(* Logix 5000 project; controller PRU vendor 1 type 14 code 107 rev 20.13; software revision 20.01; part 14 of 17 *)
(* tags used below, declared in another part *)
   AlarmMaster : DINT;
   CHANGING_TOTE_1 : BOOL;
   CSS_Status_Data : PLCStatusData;
   DailyTotalResetPB : BOOL;
   GTL1_PRESSURE_Real : REAL;
   GTL1_TEMPERATURE : DINT;
   GTL2_PRESSURE_Real : REAL;
   GTL2_TEMPERATURE : DINT;
   GTL3_PRESSURE_Real : REAL;
   GTL3_TEMPERATURE : DINT;
   IFS_CommsLoss_TMR : TIMER;   // Comms to IFS Has been Lost Alarm Timer
   IFS_CommsLossAlm : BOOL;   // Comms to IFS Has been Lost Alarm
   IFS_CommsWarning_TMR : TIMER;   // Comms to IFS Has been Lost Warning Timer
   IFS_CommsWarningAlm : BOOL;   // Comms to IFS Has been Lost Warning Alarm
   IFS_PLC_Seconds_Temp : DINT;
   IFS_Status_Data : PLCStatusData;
   IND560_Data_to_Set : SINT;
   IND560_Get_Shared_Data_Message : MESSAGE;
   IND560_Read_Data : REAL;
   IND560_Set_Shared_Data_Message : MESSAGE;
   IND560_Test_Msg : MESSAGE;
   KPI_WeightResetPB : BOOL;
   KPI_WeightResetTmr : TIMER;
   LOCAL_DATE_TIME : DateTime;
   MIDNIGHT : BOOL;
   MIDNIGHT_ONS : DINT;
   myweight_2 : DINT;
   myweight_3 : DINT;
   myweight_4 : DINT;
   OutFeedScale : SystemAlarmMonitor;
   PLC_Time : DINT[8];
   PROCESSOR_FAULT : BOOL;
   PRU_Status_Data : PLCStatusData;
   UTL_CommsLoss_TMR : TIMER;   // Comms to UTL Has been Lost Alarm Timer
   UTL_CommsLossAlm : BOOL;   // Comms to UTL Has been Lost Alarm
   UTL_CommsWarning_TMR : TIMER;   // Comms to UTL Has been Lost Warning Timer
   UTL_CommsWarningAlm : BOOL;   // Comms to UTL Has been Lost Warning Alarm
   UTL_PLC_Seconds_Temp : DINT;
   UTL_Status_Data : PLCStatusData;
   WC025_DailyTotal : REAL;
   WC025_DailyTotalLast : REAL;
   WC025_DailyTotalResetPB_ONS : BOOL;
   WC025_TareALM : BOOL;
   WEIGHT : REAL;
(* MSG, continued *)

ROUTINE IFS_MSG   (* ladder *)
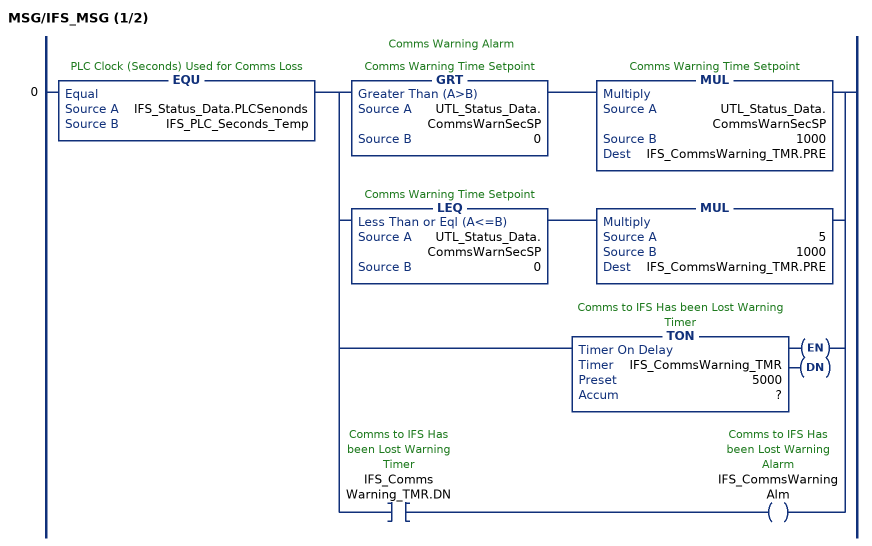
   // Comms Warning Alarm
   0: EQU(IFS_Status_Data.PLCSenonds,IFS_PLC_Seconds_Temp)[GRT(UTL_Status_Data.CommsWarnSecSP,0) MUL(UTL_Status_Data.CommsWarnSecSP,1000,IFS_CommsWarning_TMR.PRE) ,LEQ(UTL_Status_Data.CommsWarnSecSP,0) MUL(5,1000,IFS_CommsWarning_TMR.PRE) ,TON(IFS_CommsWarning_TMR,?,?) ,XIC(IFS_CommsWarning_TMR.DN) OTE(IFS_CommsWarningAlm) ];
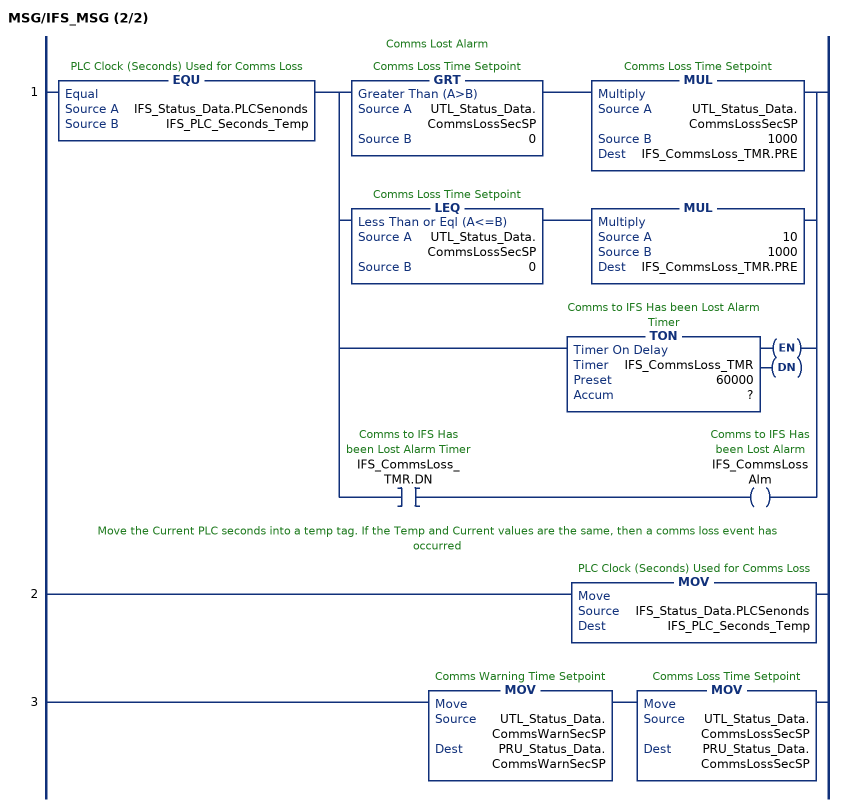
   // Comms Lost Alarm
   1: EQU(IFS_Status_Data.PLCSenonds,IFS_PLC_Seconds_Temp)[GRT(UTL_Status_Data.CommsLossSecSP,0) MUL(UTL_Status_Data.CommsLossSecSP,1000,IFS_CommsLoss_TMR.PRE) ,LEQ(UTL_Status_Data.CommsLossSecSP,0) MUL(10,1000,IFS_CommsLoss_TMR.PRE) ,TON(IFS_CommsLoss_TMR,?,?) ,XIC(IFS_CommsLoss_TMR.DN) OTE(IFS_CommsLossAlm) ];
   // Move the Current PLC seconds into a temp tag. If the Temp and Current values are the same, then a comms loss event has occurred
   2: MOV(IFS_Status_Data.PLCSenonds,IFS_PLC_Seconds_Temp);
   3: MOV(UTL_Status_Data.CommsWarnSecSP,PRU_Status_Data.CommsWarnSecSP)MOV(UTL_Status_Data.CommsLossSecSP,PRU_Status_Data.CommsLossSecSP);
END_ROUTINE

ROUTINE MSG   (* ladder *)
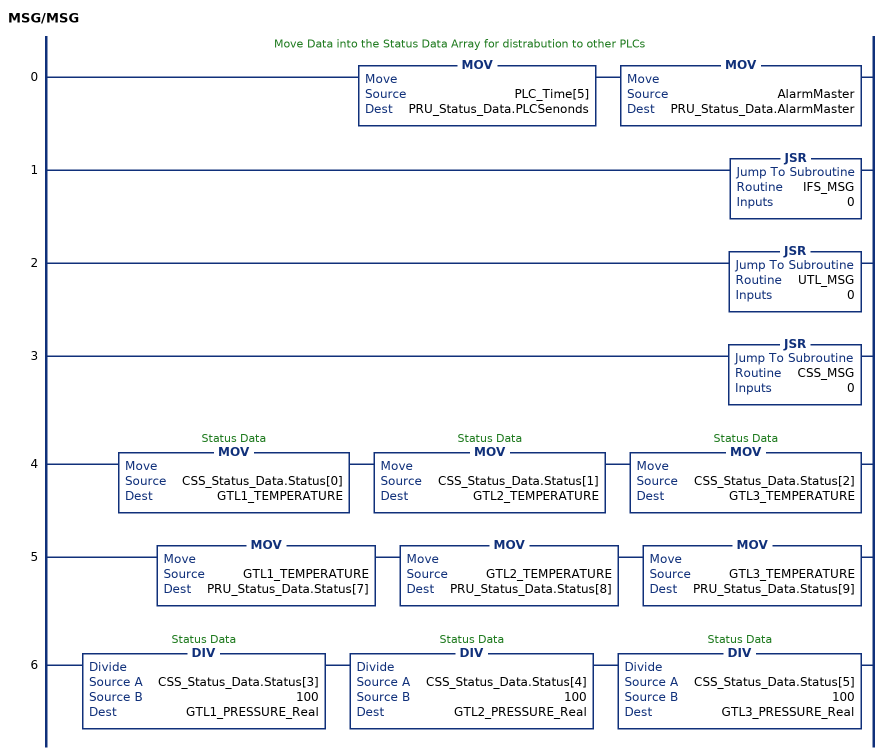
   // Move Data into the Status Data Array for distrabution to other PLCs
   0: MOV(PLC_Time[5],PRU_Status_Data.PLCSenonds)MOV(AlarmMaster,PRU_Status_Data.AlarmMaster);
   1: JSR(IFS_MSG,0);
   2: JSR(UTL_MSG,0);
   3: JSR(CSS_MSG,0);
   4: MOV(CSS_Status_Data.Status[0],GTL1_TEMPERATURE)MOV(CSS_Status_Data.Status[1],GTL2_TEMPERATURE)MOV(CSS_Status_Data.Status[2],GTL3_TEMPERATURE);
   5: MOV(GTL1_TEMPERATURE,PRU_Status_Data.Status[7])MOV(GTL2_TEMPERATURE,PRU_Status_Data.Status[8])MOV(GTL3_TEMPERATURE,PRU_Status_Data.Status[9]);
   6: DIV(CSS_Status_Data.Status[3],100,GTL1_PRESSURE_Real)DIV(CSS_Status_Data.Status[4],100,GTL2_PRESSURE_Real)DIV(CSS_Status_Data.Status[5],100,GTL3_PRESSURE_Real);
END_ROUTINE

ROUTINE UTL_MSG   (* ladder *)
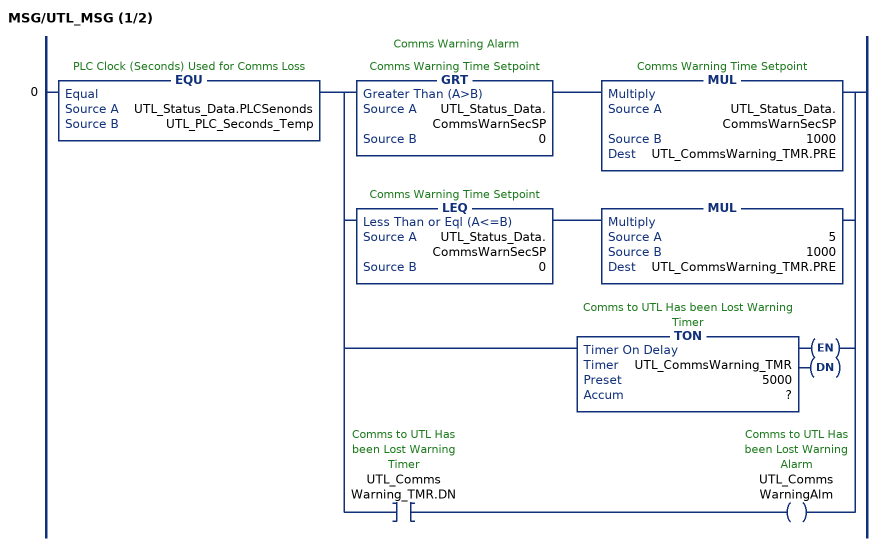
   // Comms Warning Alarm
   0: EQU(UTL_Status_Data.PLCSenonds,UTL_PLC_Seconds_Temp)[GRT(UTL_Status_Data.CommsWarnSecSP,0) MUL(UTL_Status_Data.CommsWarnSecSP,1000,UTL_CommsWarning_TMR.PRE) ,LEQ(UTL_Status_Data.CommsWarnSecSP,0) MUL(5,1000,UTL_CommsWarning_TMR.PRE) ,TON(UTL_CommsWarning_TMR,?,?) ,XIC(UTL_CommsWarning_TMR.DN) OTE(UTL_CommsWarningAlm) ];
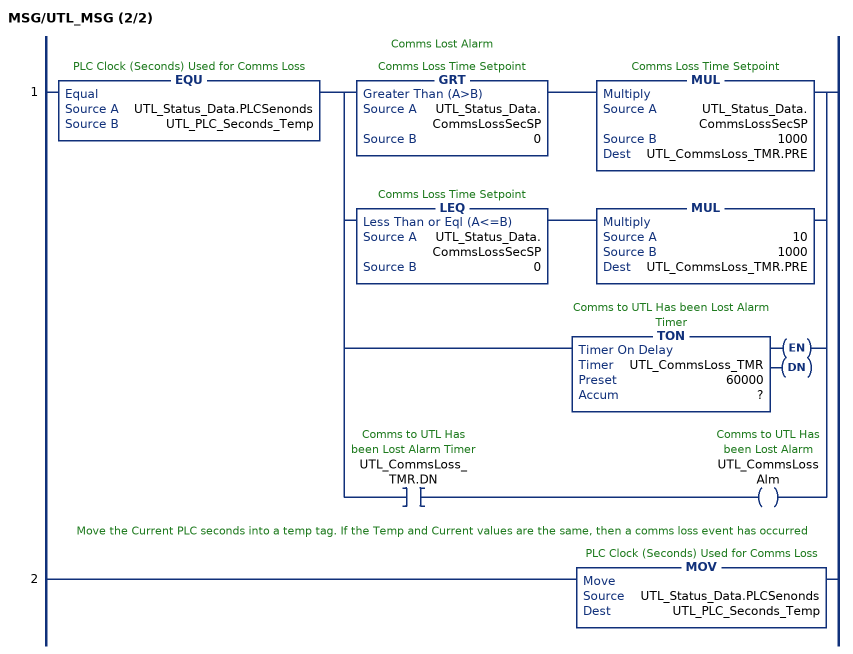
   // Comms Lost Alarm
   1: EQU(UTL_Status_Data.PLCSenonds,UTL_PLC_Seconds_Temp)[GRT(UTL_Status_Data.CommsLossSecSP,0) MUL(UTL_Status_Data.CommsLossSecSP,1000,UTL_CommsLoss_TMR.PRE) ,LEQ(UTL_Status_Data.CommsLossSecSP,0) MUL(10,1000,UTL_CommsLoss_TMR.PRE) ,TON(UTL_CommsLoss_TMR,?,?) ,XIC(UTL_CommsLoss_TMR.DN) OTE(UTL_CommsLossAlm) ];
   // Move the Current PLC seconds into a temp tag. If the Temp and Current values are the same, then a comms loss event has occurred
   2: MOV(UTL_Status_Data.PLCSenonds,UTL_PLC_Seconds_Temp);
END_ROUTINE
END_PROGRAM

PROGRAM Never_Fault_Logic   (* main routine Main *)
VAR
   HMI_CONTROLLER_DISPLAY : MAJOR_FAULT := (TYPE := 4, CODE := 20, INFO[0] := 2, INFO[1] := 46883, INFO[2] := 46883, INFO[3] := 1637264, INFO[4] := 1989688);
   MAJORFAULT_RECORD : FAULTRECORD;
END_VAR

ROUTINE Main   (* ladder *)
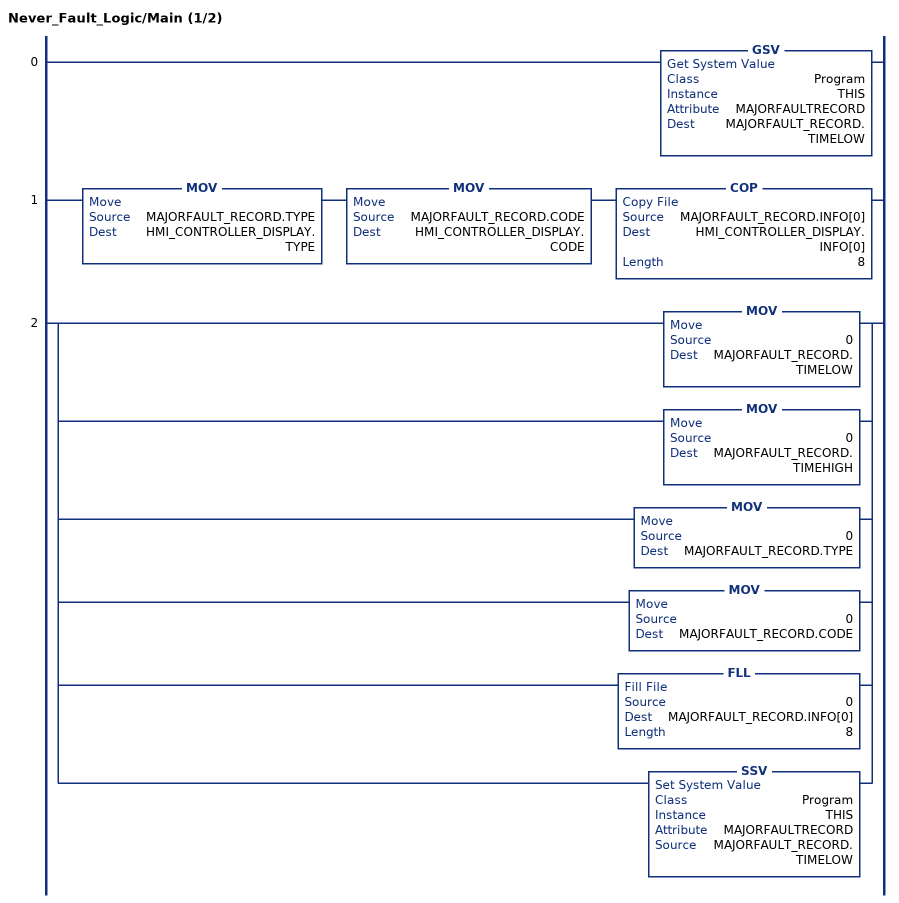
   0: GSV(Program,THIS,MAJORFAULTRECORD,MAJORFAULT_RECORD.TIMELOW);
   1: MOV(MAJORFAULT_RECORD.TYPE,HMI_CONTROLLER_DISPLAY.TYPE)MOV(MAJORFAULT_RECORD.CODE,HMI_CONTROLLER_DISPLAY.CODE)COP(MAJORFAULT_RECORD.INFO[0],HMI_CONTROLLER_DISPLAY.INFO[0],8);
   2: [MOV(0,MAJORFAULT_RECORD.TIMELOW) ,MOV(0,MAJORFAULT_RECORD.TIMEHIGH) ,MOV(0,MAJORFAULT_RECORD.TYPE) ,MOV(0,MAJORFAULT_RECORD.CODE) ,FLL(0,MAJORFAULT_RECORD.INFO[0],8) ,SSV(Program,THIS,MAJORFAULTRECORD,MAJORFAULT_RECORD.TIMELOW) ];
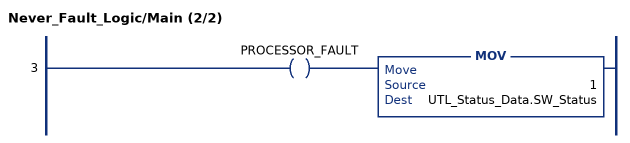
   3: OTE(PROCESSOR_FAULT)MOV(1,UTL_Status_Data.SW_Status);
END_ROUTINE
END_PROGRAM

PROGRAM OutFeedScale   (* main routine MainRoutine *)
VAR
   AlarmMasterResetTON : TIMER := (PRE := 1000, ACC := 676, EN := 1, TT := 1);
   AlarmsAckAll : BOOL;
   AlarmsDisabled : BOOL;
   EmptyToteWeight : REAL := 5.0;
   Get_Data : BOOL;
   Gotten_Data : REAL;
   Gotton_Data : REAL;
   IND560_Get_Shared_Data_MessageONS : BOOL;
   IND560_GetDataTmr : TIMER := (PRE := 1000);
   IND560_GetDataTmrSecSP : DINT := 1;
   IND560_NetWeightLbs : REAL;
   LoadTargetTmr : TIMER := (PRE := 2000);
   Major : DINT := 6;
   Minor : DINT;
   MyGet : BOOL;
   myweight : DINT := 65463;
   OutFeed_AlarmMaster : DINT;
   OutFeed_WC025_CommsErrorSec : DINT;
   OutFeed_WC025_CommsLossSec : DINT;
   OutFeed_WC025_EntryStatus : DINT;
   Revision : DINT;
   Set_Data : BOOL;
   Slot_1_Weight : REAL;
   Slot_2_Weight : REAL := 45312.0;
   Slot_3_Weight : REAL := 65463.0;
   Slot_4_Weight : REAL := 45312.0;
   TarePB : BOOL;
   testchar : REAL := 12.0;
   WC025 : AnalogControl := (AUTO := 1, HHEnabled := 1, HEnabled := 1);
   WC025_AddONS1 : BOOL;
   WC025_Alm : ALARM_ANALOG;
   WC025_BatchTotal : DINT;
   WC025_CommsErrorAlm : BOOL;
   WC025_CommsErrorTmr : TIMER;
   WC025_CommsLossAlm : BOOL;
   WC025_CommsLossTmr : TIMER;
   WC025_CummulativeTotal : DINT;
   WC025_EntryStatus : DINT := 16384;
   WC025_EntryStatusSint : SINT := 4;
   WC025_Full : BOOL;
   WC025_Full_TON : TIMER := (PRE := 5000);
   WC025_FullDiffSP : REAL := 896.0;
   WC025_FullSP : REAL := 901.0;
   WC025_PV_Add : REAL;
   WC025_PV_AddDB : REAL := 0.1;
   WC025_PV_Last : REAL;
   WC025_SwapONS : BOOL;
   WC025_SwapONS1 : BOOL;
   WC025_SwapONS2 : BOOL := 1;
   WC025_SwapPB : BOOL := 1;
   WC025_Total : REAL;
   WC025_TotalLast : REAL;
   WC025_TotalResetPB : BOOL;
   WC025_ToteTotal : REAL;
END_VAR

ROUTINE A0_Serialize_Me   (* ladder *)
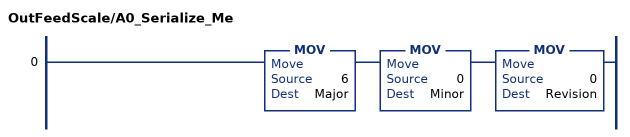
   0: MOV(6,Major)MOV(0,Minor)MOV(0,Revision);
END_ROUTINE

ROUTINE A5_AlarmMaster   (* ladder *)
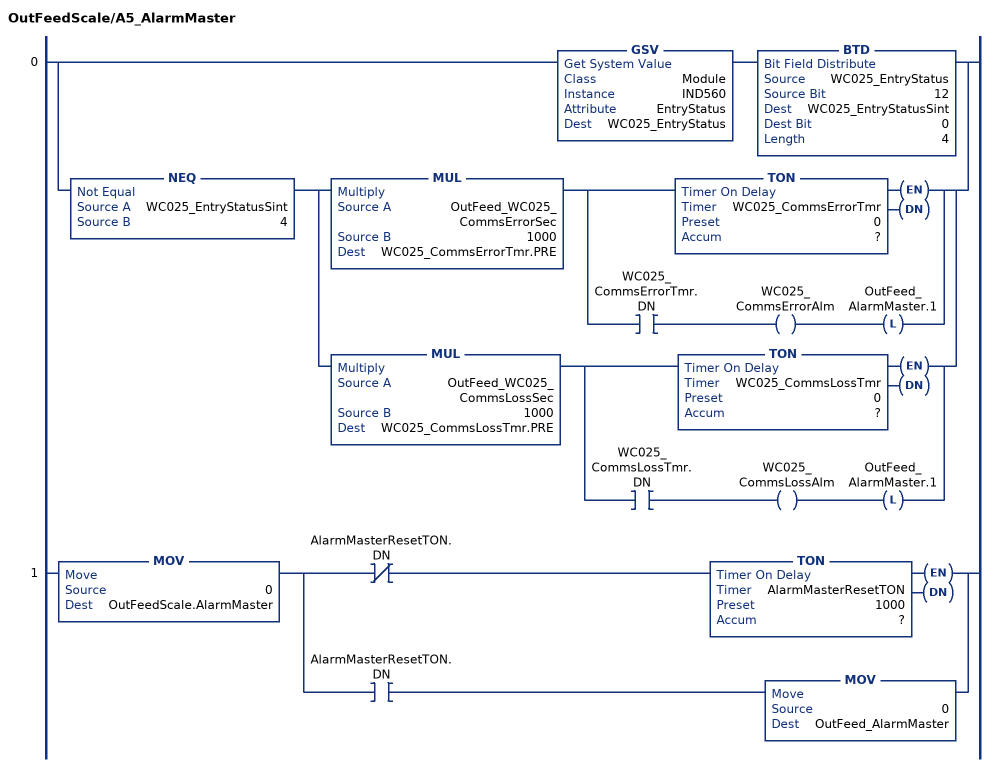
   0: [GSV(Module,IND560,EntryStatus,WC025_EntryStatus) BTD(WC025_EntryStatus,12,WC025_EntryStatusSint,0,4) ,NEQ(WC025_EntryStatusSint,4) [MUL(OutFeed_WC025_CommsErrorSec,1000,WC025_CommsErrorTmr.PRE) [TON(WC025_CommsErrorTmr,?,?) ,XIC(WC025_CommsErrorTmr.DN) OTE(WC025_CommsErrorAlm) OTL(OutFeed_AlarmMaster.1) ] ,MUL(OutFeed_WC025_CommsLossSec,1000,WC025_CommsLossTmr.PRE) [TON(WC025_CommsLossTmr,?,?) ,XIC(WC025_CommsLossTmr.DN) OTE(WC025_CommsLossAlm) OTL(OutFeed_AlarmMaster.1) ] ] ];
   1: MOV(0,OutFeedScale.AlarmMaster)[XIO(AlarmMasterResetTON.DN) TON(AlarmMasterResetTON,?,?) ,XIC(AlarmMasterResetTON.DN) MOV(0,OutFeed_AlarmMaster) ];
END_ROUTINE

ROUTINE MainRoutine   (* ladder *)
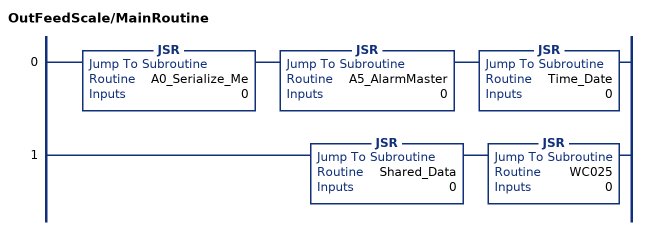
   0: JSR(A0_Serialize_Me,0)JSR(A5_AlarmMaster,0)JSR(Time_Date,0);
   1: JSR(Shared_Data,0)JSR(WC025,0);
END_ROUTINE

ROUTINE Shared_Data   (* ladder *)
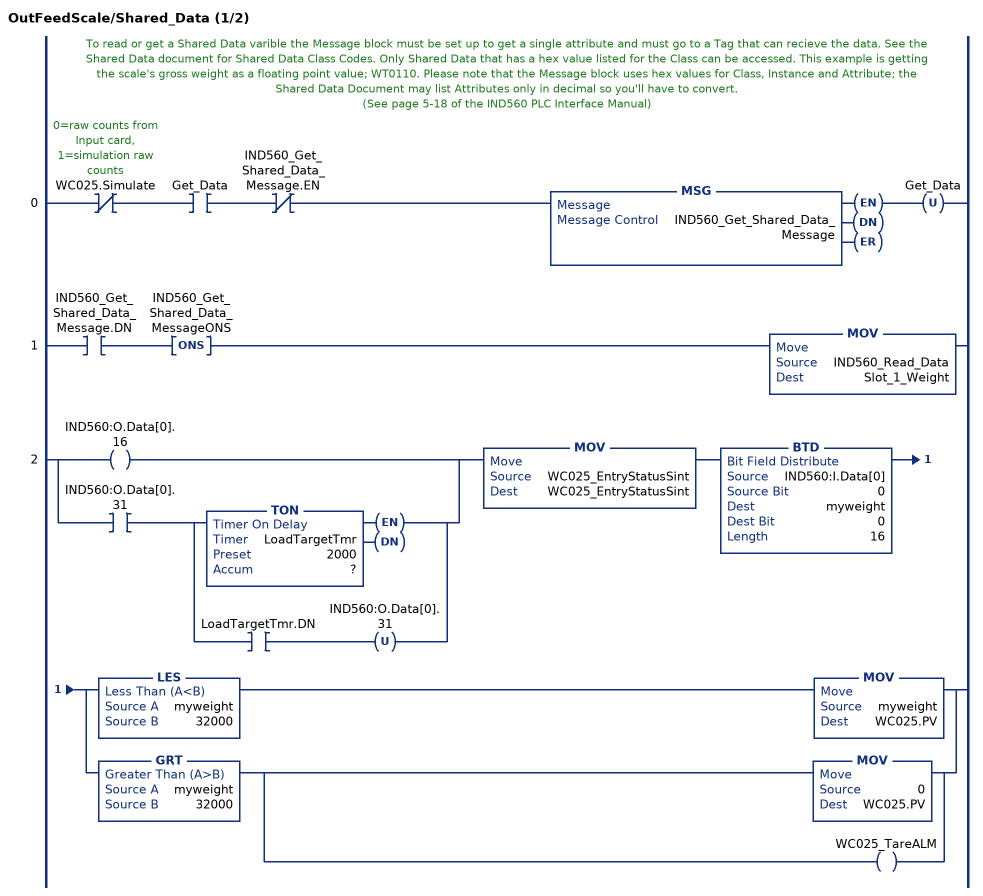
   // To read or get a Shared Data varible the Message block must be set up to get a single attribute and must go to a Tag that can recieve the data. See the Shared Data document for Shared Data Class Codes. Only Shared Data that has a hex value listed for the Class can be accessed. This example is getting the scale's gross weight as a floating point value; WT0110. Please note that the Message block uses hex values for Class, Instance and Attribute; the Shared Data Document may list Attributes only in decimal so you'll have to convert.
   // (See page 5-18 of the IND560 PLC Interface Manual)
   0: XIO(WC025.Simulate)XIC(Get_Data)XIO(IND560_Get_Shared_Data_Message.EN)MSG(IND560_Get_Shared_Data_Message)OTU(Get_Data);
   1: XIC(IND560_Get_Shared_Data_Message.DN)ONS(IND560_Get_Shared_Data_MessageONS)MOV(IND560_Read_Data,Slot_1_Weight);
   2: [OTE(IND560:O.Data[0].16) ,XIC(IND560:O.Data[0].31) [TON(LoadTargetTmr,?,?) ,XIC(LoadTargetTmr.DN) OTU(IND560:O.Data[0].31) ] ]MOV(WC025_EntryStatusSint,WC025_EntryStatusSint)BTD(IND560:I.Data[0],0,myweight,0,16)[LES(myweight,32000) MOV(myweight,WC025.PV) ,GRT(myweight,32000) [MOV(0,WC025.PV) ,OTE(WC025_TareALM) ] ];
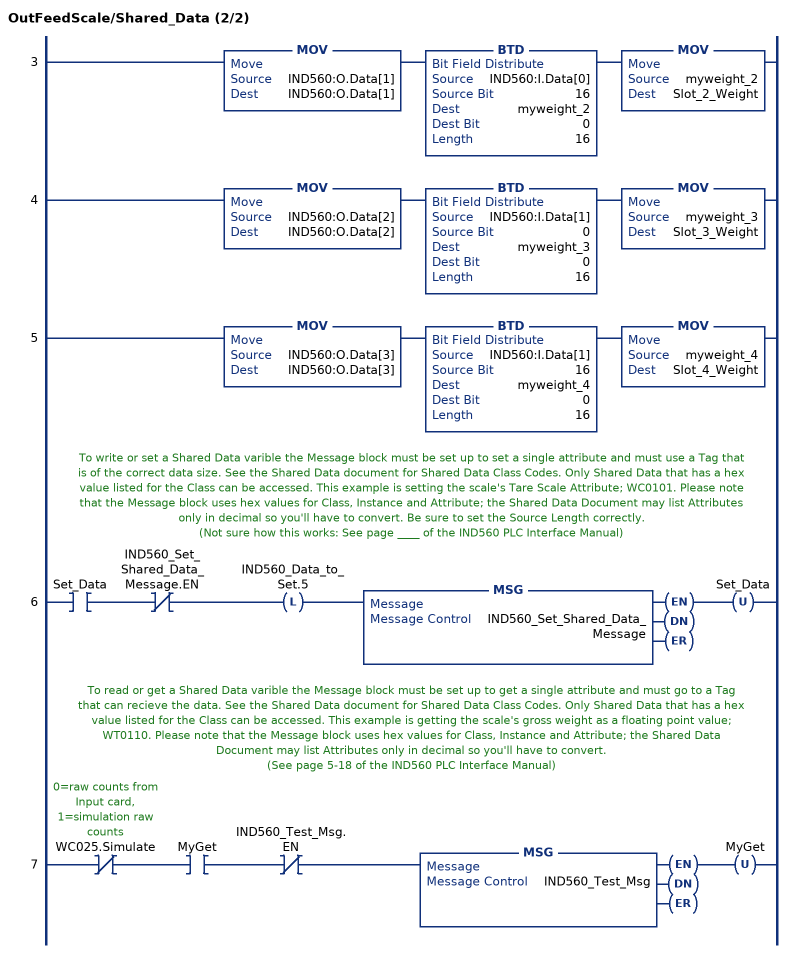
   3: MOV(IND560:O.Data[1],IND560:O.Data[1])BTD(IND560:I.Data[0],16,myweight_2,0,16)MOV(myweight_2,Slot_2_Weight);
   4: MOV(IND560:O.Data[2],IND560:O.Data[2])BTD(IND560:I.Data[1],0,myweight_3,0,16)MOV(myweight_3,Slot_3_Weight);
   5: MOV(IND560:O.Data[3],IND560:O.Data[3])BTD(IND560:I.Data[1],16,myweight_4,0,16)MOV(myweight_4,Slot_4_Weight);
   // To write or set a Shared Data varible the Message block must be set up to set a single attribute and must use a Tag that is of the correct data size. See the Shared Data document for Shared Data Class Codes. Only Shared Data that has a hex value listed for the Class can be accessed. This example is setting the scale's Tare Scale Attribute; WC0101. Please note that the Message block uses hex values for Class, Instance and Attribute; the Shared Data Document may list Attributes only in decimal so you'll have to convert. Be sure to set the Source Length correctly.
   // (Not sure how this works: See page ____ of the IND560 PLC Interface Manual)
   6: XIC(Set_Data)XIO(IND560_Set_Shared_Data_Message.EN)OTL(IND560_Data_to_Set.5)MSG(IND560_Set_Shared_Data_Message)OTU(Set_Data);
   // To read or get a Shared Data varible the Message block must be set up to get a single attribute and must go to a Tag that can recieve the data. See the Shared Data document for Shared Data Class Codes. Only Shared Data that has a hex value listed for the Class can be accessed. This example is getting the scale's gross weight as a floating point value; WT0110. Please note that the Message block uses hex values for Class, Instance and Attribute; the Shared Data Document may list Attributes only in decimal so you'll have to convert.
   // (See page 5-18 of the IND560 PLC Interface Manual)
   7: XIO(WC025.Simulate)XIC(MyGet)XIO(IND560_Test_Msg.EN)MSG(IND560_Test_Msg)OTU(MyGet);
END_ROUTINE

ROUTINE Time_Date   (* ladder *)
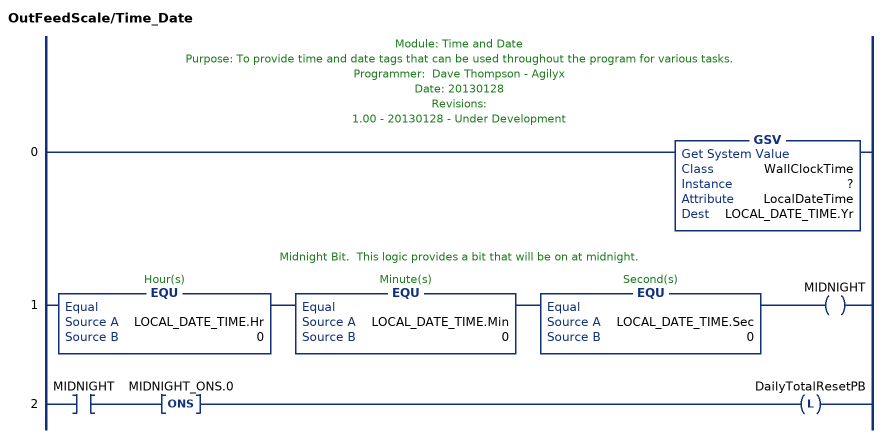
   // Module: Time and Date
   // Purpose: To provide time and date tags that can be used throughout the program for various tasks.
   // Programmer:  Dave Thompson - Agilyx
   // Date: 20130128
   // Revisions:
   // 1.00 - 20130128 - Under Development
   0: GSV(WallClockTime,?,LocalDateTime,LOCAL_DATE_TIME.Yr);
   // Midnight Bit.  This logic provides a bit that will be on at midnight.
   1: EQU(LOCAL_DATE_TIME.Hr,0)EQU(LOCAL_DATE_TIME.Min,0)EQU(LOCAL_DATE_TIME.Sec,0)OTE(MIDNIGHT);
   2: XIC(MIDNIGHT)ONS(MIDNIGHT_ONS.0)OTL(DailyTotalResetPB);
END_ROUTINE

ROUTINE WC025   (* ladder *)
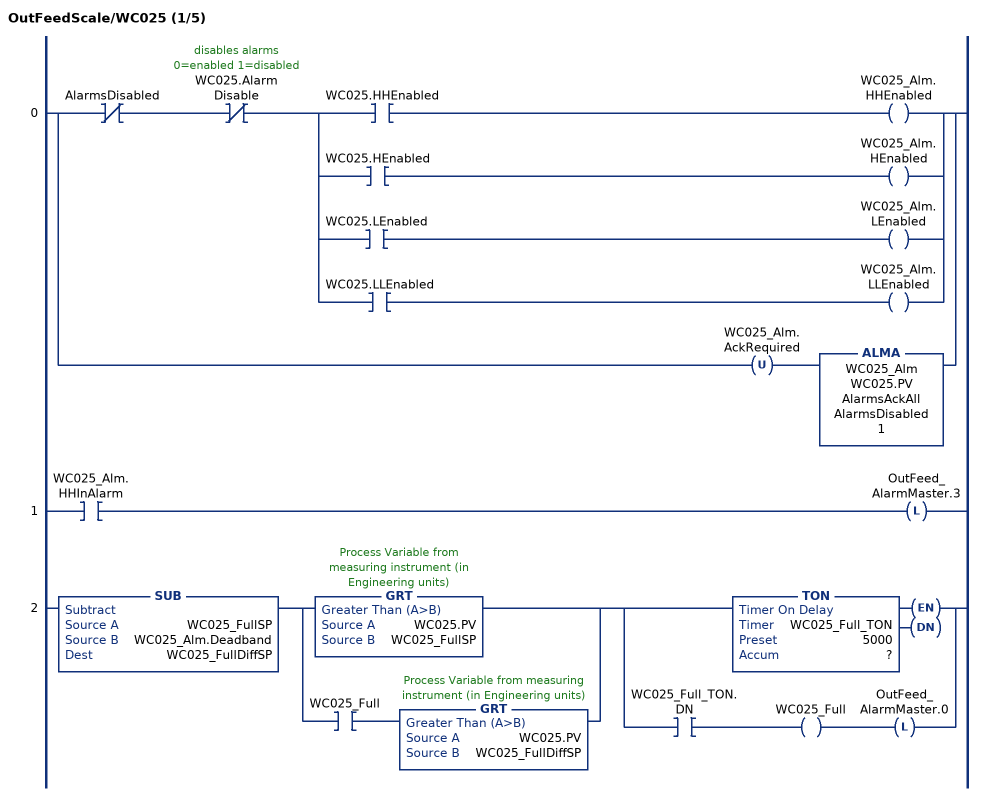
   0: [XIO(AlarmsDisabled) XIO(WC025.AlarmDisable) [XIC(WC025.HHEnabled) OTE(WC025_Alm.HHEnabled) ,XIC(WC025.HEnabled) OTE(WC025_Alm.HEnabled) ,XIC(WC025.LEnabled) OTE(WC025_Alm.LEnabled) ,XIC(WC025.LLEnabled) OTE(WC025_Alm.LLEnabled) ] ,OTU(WC025_Alm.AckRequired) ALMA(WC025_Alm,WC025.PV,AlarmsAckAll,AlarmsDisabled,1) ];
   1: XIC(WC025_Alm.HHInAlarm)OTL(OutFeed_AlarmMaster.3);
   2: SUB(WC025_FullSP,WC025_Alm.Deadband,WC025_FullDiffSP)[GRT(WC025.PV,WC025_FullSP) ,XIC(WC025_Full) GRT(WC025.PV,WC025_FullDiffSP) ][TON(WC025_Full_TON,?,?) ,XIC(WC025_Full_TON.DN) OTE(WC025_Full) OTL(OutFeed_AlarmMaster.0) ];
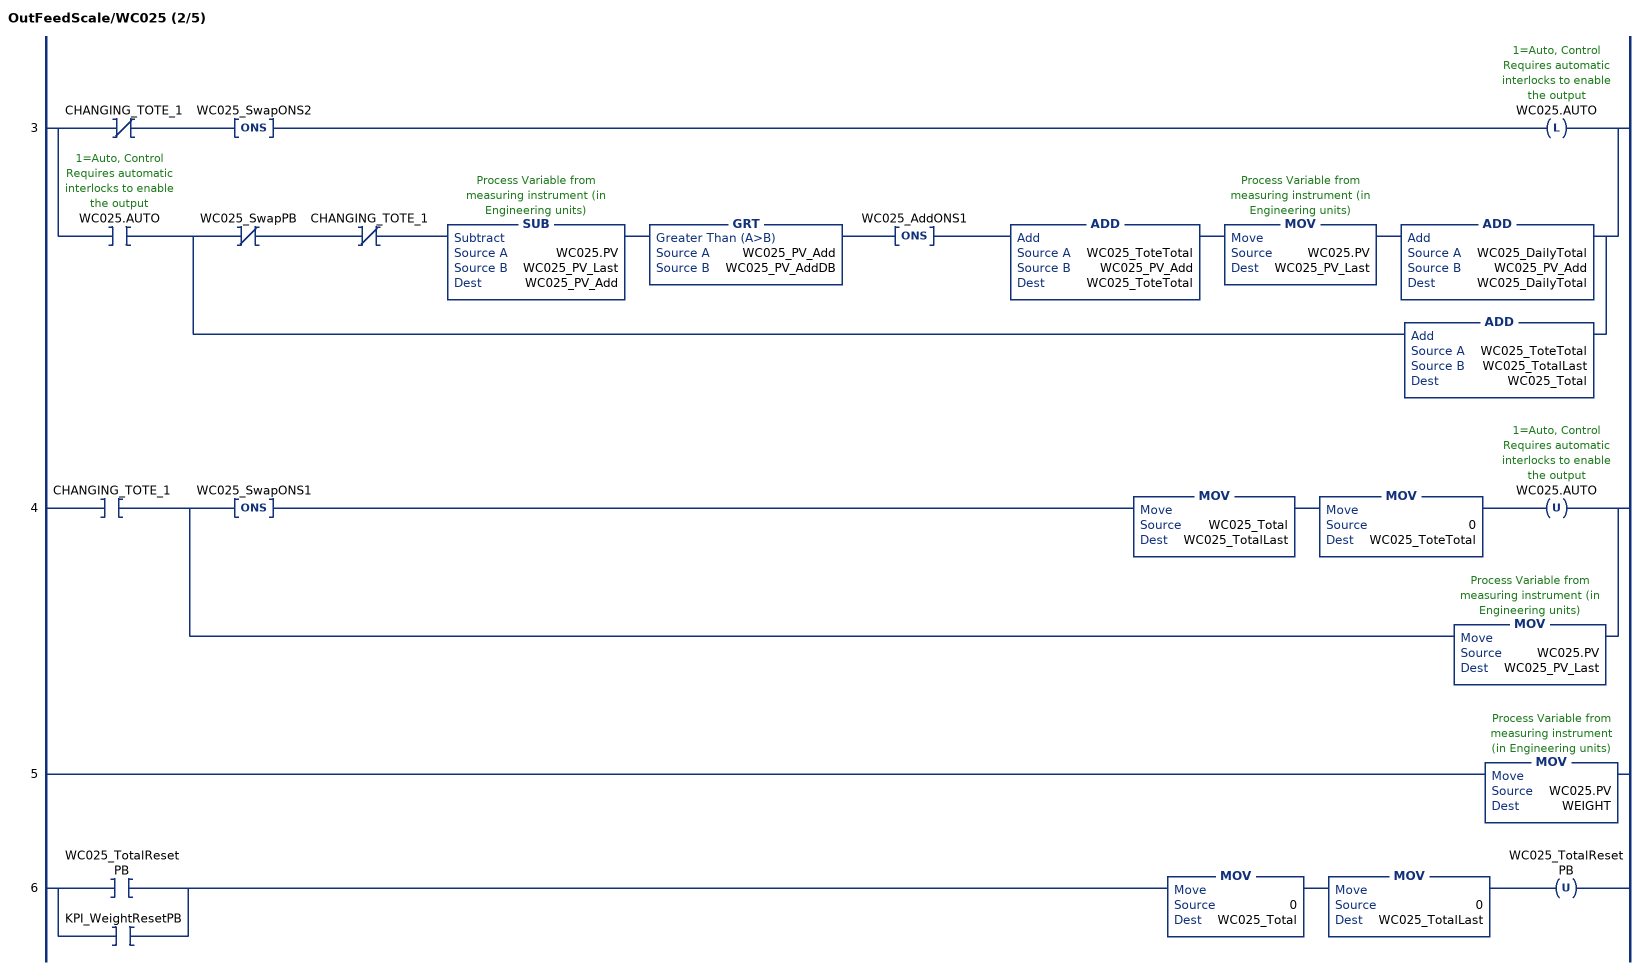
   3: [XIO(CHANGING_TOTE_1) ONS(WC025_SwapONS2) OTL(WC025.AUTO) ,XIC(WC025.AUTO) [XIO(WC025_SwapPB) XIO(CHANGING_TOTE_1) SUB(WC025.PV,WC025_PV_Last,WC025_PV_Add) GRT(WC025_PV_Add,WC025_PV_AddDB) ONS(WC025_AddONS1) ADD(WC025_ToteTotal,WC025_PV_Add,WC025_ToteTotal) MOV(WC025.PV,WC025_PV_Last) ADD(WC025_DailyTotal,WC025_PV_Add,WC025_DailyTotal) ,ADD(WC025_ToteTotal,WC025_TotalLast,WC025_Total) ] ];
   4: XIC(CHANGING_TOTE_1)[ONS(WC025_SwapONS1) MOV(WC025_Total,WC025_TotalLast) MOV(0,WC025_ToteTotal) OTU(WC025.AUTO) ,MOV(WC025.PV,WC025_PV_Last) ];
   5: MOV(WC025.PV,WEIGHT);
   6: [XIC(WC025_TotalResetPB) ,XIC(KPI_WeightResetPB) ]MOV(0,WC025_Total)MOV(0,WC025_TotalLast)OTU(WC025_TotalResetPB);
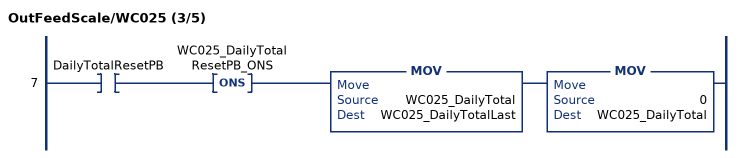
   7: XIC(DailyTotalResetPB)ONS(WC025_DailyTotalResetPB_ONS)MOV(WC025_DailyTotal,WC025_DailyTotalLast)MOV(0,WC025_DailyTotal);
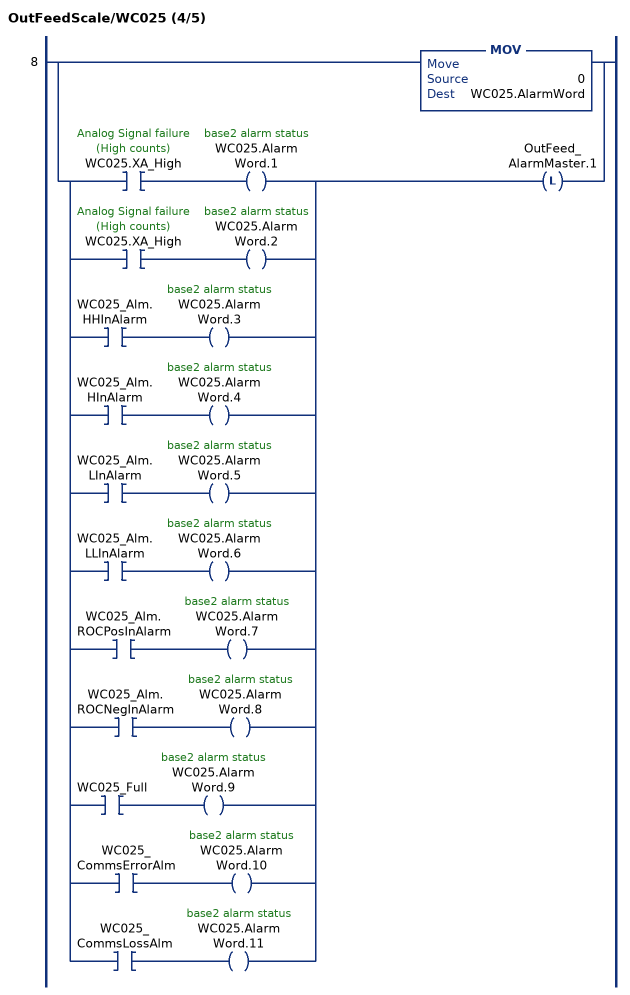
   8: [MOV(0,WC025.AlarmWord) ,[XIC(WC025.XA_High) OTE(WC025.AlarmWord.1) ,XIC(WC025.XA_High) OTE(WC025.AlarmWord.2) ,XIC(WC025_Alm.HHInAlarm) OTE(WC025.AlarmWord.3) ,XIC(WC025_Alm.HInAlarm) OTE(WC025.AlarmWord.4) ,XIC(WC025_Alm.LInAlarm) OTE(WC025.AlarmWord.5) ,XIC(WC025_Alm.LLInAlarm) OTE(WC025.AlarmWord.6) ,XIC(WC025_Alm.ROCPosInAlarm) OTE(WC025.AlarmWord.7) ,XIC(WC025_Alm.ROCNegInAlarm) OTE(WC025.AlarmWord.8) ,XIC(WC025_Full) OTE(WC025.AlarmWord.9) ,XIC(WC025_CommsErrorAlm) OTE(WC025.AlarmWord.10) ,XIC(WC025_CommsLossAlm) OTE(WC025.AlarmWord.11) ] OTL(OutFeed_AlarmMaster.1) ];
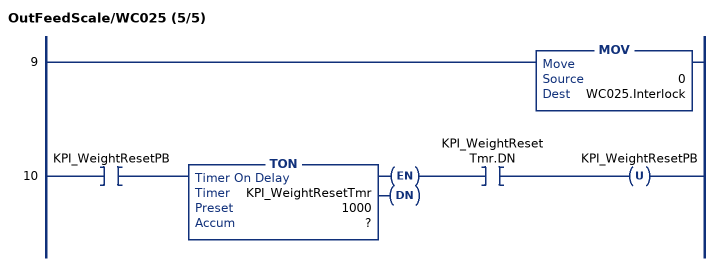
   9: MOV(0,WC025.Interlock);
   10: XIC(KPI_WeightResetPB)TON(KPI_WeightResetTmr,?,?)XIC(KPI_WeightResetTmr.DN)OTU(KPI_WeightResetPB);
END_ROUTINE
END_PROGRAM
